TYPE FB_LaserScannerR2000_Antwort :
STRUCT
	handle : STRING(20);
	error_code : DINT;
	error_text : STRING(255);
END_STRUCT
END_TYPE

(* stored: Version 1.1.0.1, ProductVersion 3.1.4018.5
   DUT FB_LaserScannerR2000_Antwort: Id {3d727c2a-c36f-4bc9-85b1-2d00c6e8e7da} *)
